PROGRAM AutoStates_POU
VAR
END_VAR

END_PROGRAM

(* stored: Version 1.1.0.1, ProductVersion 3.1.4024.0
   POU AutoStates_POU: Id {b3a9f5a3-18ec-404a-a269-7e864e0ccca1}, SpecialFunc None *)
